RoboDK station: Larry_Station.rdk

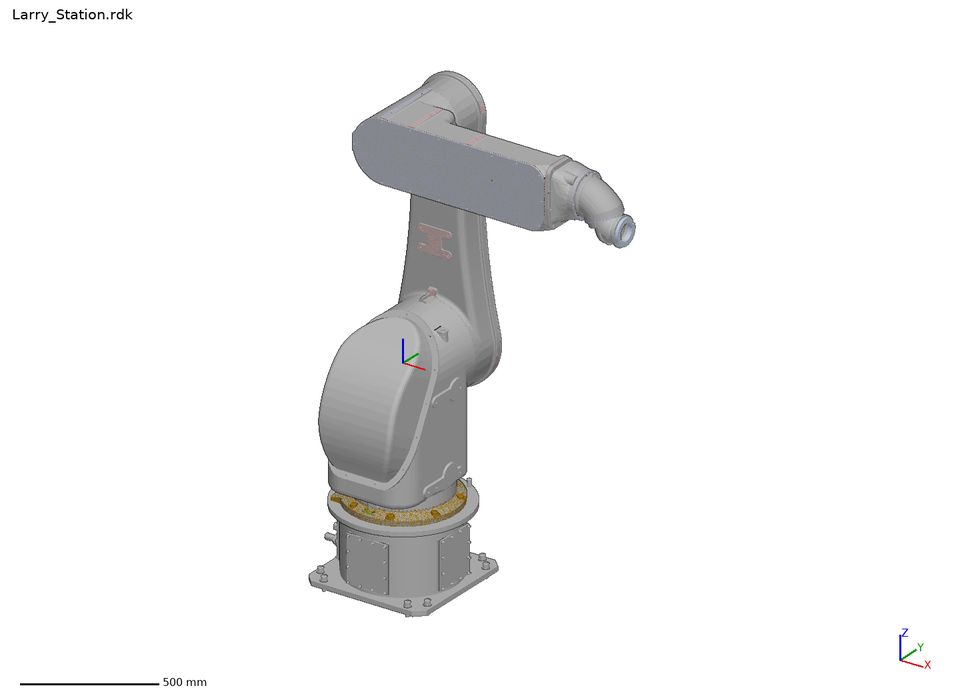
[picture v0: the station drawn from its stored meshes, robots at their saved joint values, targets as dots, program paths as lines]
Station Larry_Station (saved by RoboDK 5.5.4). Poses are relative to the parent item; angles as X-Y-Z fixed-axis rotations.
Station parameters (name, value as stored): LIN64
  - frame Fanuc P-50iB/10L Base at (0, 0, 850) mm
    - robot Fanuc P-50iB/10L: 6 axes, payload 10 kg, reach 1800 mm, repeatability 0.2 mm, weight 331 kg
        modified DH rows (alpha deg, a mm, theta deg, d mm): 0, 0, 0, 850; -90, 0, -90, 0; 0, 900, 0, 0; -90, 0, -90, 863.603; 70, 0, 0, 106.418; -70, 0, 0, 82
        base shift (0, 0, -850) mm
        joint limits [-160, -45, -205, -360, -360, -360] to [160, 120, 165, 360, 360, 360]; home [0, 0, 0, 0, 0, 0]; saved at [0, 0, 0, 0, 0, 0]
